Fanuc KAREL source: ko00149.KL

-- PROVISIONAL review KL for V940-1; original PC SHA256 c20b3b588d2479280d445791483e8e04921b04296768117feb8e6f729d68e1ec
-- Incomplete behavior may be omitted. Consult companion uncertainty JSON. Do not deploy.
PROGRAM KO00149
%NOLOCKGROUP
VAR
  R : REAL
  N : INTEGER
-- UNRESOLVED_DECL CFG type=00001c
-- UNRESOLVED_DECL OUT type=000102
BEGIN
  -- V9_ZERO_TABLE_METADATA_HINT layout=0001; no indexed target words; source/name/runtime held
  -- UNRESOLVED_PC offsets 5-12; opcodes 9D,23
  -- UNRESOLVED_PC offsets 17-28; opcodes 2E,23
  -- UNRESOLVED_PC offsets 33-43; opcodes 9D,22,A5
  -- UNRESOLVED_PC offsets 48-107; opcodes 27,22,22,22,22,22,27,21,64,22,76,7E,4A
  -- UNRESOLVED_PC offsets 112-116; opcodes 7F
END KO00149
